// SIMATIC STEP 7 (V5.x) project Q6
// CPU: CPU 313C
// station: Hardware
// station: SIMATIC 300(1)
// station: P_ADR_BUS
// program: S7 Program(1)

SYMBOL_TABLE
"Counter"	C 0	COUNTER
"SCALE"	FC 105	FC 105	// Scaling Values
"UNSCALE"	FC 106	FC 106	// Unscaling Values
"Start"	I 0.0	BOOL
"Stop"	I 0.1	BOOL
"Input Thermocouple"	ID 20	REAL
"Bipolar scale/unscale"	M 0.0	BOOL
"Reserve Motor mem"	M 0.1	BOOL
"MD20"	MD 20	REAL
"Temp INPUT"	MD 30	REAL
"Round Temp INPUT"	MD 50	DINT
"Counter num"	MW 3	INT
"Error Unscale"	MW 10	WORD
"Error Scale"	MW 11	WORD
"Memory OUTPUT"	MW 40	INT
"Buffer"	MW 45	INT
"Out Unscale/IN Scale"	MW 100	INT
"Motor 1"	Q 0.0	BOOL
"Reserve Motor"	Q 0.1	BOOL
"QW100"	QW 100	INT
"Timer"	T 0	TIMER
END_SYMBOL_TABLE

// FC 105: know-how protected block, not included

// FC 106: know-how protected block, not included

ORGANIZATION_BLOCK OB 1
TITLE = "Main Program Sweep (Cycle)"
VERSION : 0.1
VAR_TEMP
  OB1_EV_CLASS : BYTE ;	//Bits 0-3 = 1 (Coming event), Bits 4-7 = 1 (Event class 1)
  OB1_SCAN_1 : BYTE ;	//1 (Cold restart scan 1 of OB 1), 3 (Scan 2-n of OB 1)
  OB1_PRIORITY : BYTE ;	//Priority of OB Execution
  OB1_OB_NUMBR : BYTE ;	//1 (Organization block 1, OB1)
  OB1_RESERVED_1 : BYTE ;	//Reserved for system
  OB1_RESERVED_2 : BYTE ;	//Reserved for system
  OB1_PREV_CYCLE : INT ;	//Cycle time of previous OB1 scan (milliseconds)
  OB1_MIN_CYCLE : INT ;	//Minimum cycle time of OB1 (milliseconds)
  OB1_MAX_CYCLE : INT ;	//Maximum cycle time of OB1 (milliseconds)
  OB1_DATE_TIME : DATE_AND_TIME ;	//Date and time OB1 started
END_VAR
BEGIN
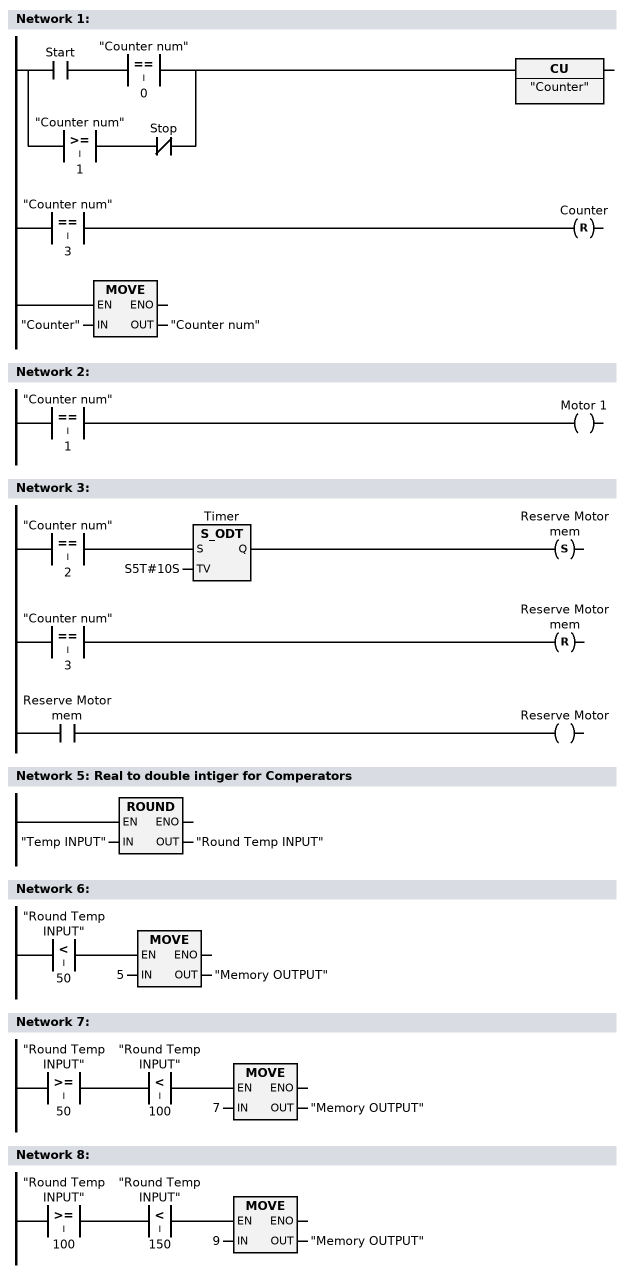
NETWORK
TITLE =
      A(;
      A     "Start";
      A(;
      L     "Counter num";
      L     0;
      ==I;
      );
      O;
      A(;
      L     "Counter num";
      L     1;
      >=I;
      );
      AN    "Stop";
      );
      CU    "Counter";
      BLD   101;
      NOP   0;
      NOP   0;
      A(;
      L     "Counter num";
      L     3;
      ==I;
      );
      R     "Counter";
      L     "Counter";
      T     "Counter num";
      NOP   0;
      NOP   0;
NETWORK
TITLE =
      L     "Counter num";
      L     1;
      ==I;
      =     "Motor 1";
NETWORK
TITLE =
      A(;
      A(;
      L     "Counter num";
      L     2;
      ==I;
      );
      L     S5T#10S;
      SD    "Timer";
      NOP   0;
      NOP   0;
      NOP   0;
      A     "Timer";
      );
      S     "Reserve Motor mem";
      A(;
      L     "Counter num";
      L     3;
      ==I;
      );
      R     "Reserve Motor mem";
      A     "Reserve Motor mem";
      =     "Reserve Motor";
NETWORK
TITLE =
      A     "Bipolar scale/unscale";
      =     L 20.0;
      BLD   103;
      A(;
      A     "Bipolar scale/unscale";
      =     L 20.1;
      BLD   103;
      CALL  "UNSCALE" (
           $1                       := "Input Thermocouple",
           $2                       := L#1101004800,
           $3                       := L#1082130432,
           $4                       := L 20.1,
           $5                       := "Error Unscale",
           $6                       := "Out Unscale/IN Scale");
      A     BR;
      );
      JNB   _001;
      CALL  "SCALE" (
           $1                       := "Out Unscale/IN Scale",
           $2                       := L#1148846080,
           $3                       := L#-1027080192,
           $4                       := L 20.0,
           $5                       := "Error Scale",
           $6                       := "Temp INPUT");
_001: NOP   0;
NETWORK
TITLE = Real to double intiger for Comperators
      L     "Temp INPUT";
      RND;
      T     "Round Temp INPUT";
      NOP   0;
NETWORK
TITLE =
      A(;
      L     "Round Temp INPUT";
      L     50;
      <I;
      );
      JNB   _002;
      L     5;
      T     "Memory OUTPUT";
_002: NOP   0;
NETWORK
TITLE =
      A(;
      L     "Round Temp INPUT";
      L     50;
      >=I;
      );
      A(;
      L     "Round Temp INPUT";
      L     100;
      <I;
      );
      JNB   _003;
      L     7;
      T     "Memory OUTPUT";
_003: NOP   0;
NETWORK
TITLE =
      A(;
      L     "Round Temp INPUT";
      L     100;
      >=I;
      );
      A(;
      L     "Round Temp INPUT";
      L     150;
      <I;
      );
      JNB   _004;
      L     9;
      T     "Memory OUTPUT";
_004: NOP   0;
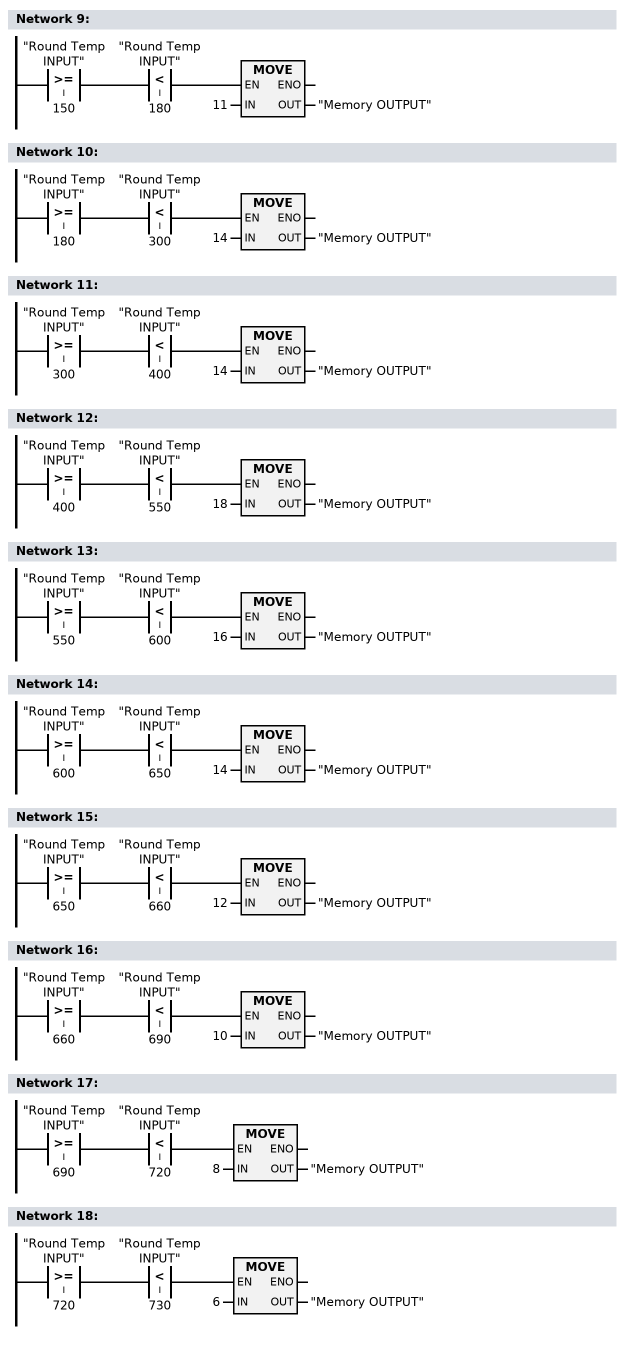
NETWORK
TITLE =
      A(;
      L     "Round Temp INPUT";
      L     150;
      >=I;
      );
      A(;
      L     "Round Temp INPUT";
      L     180;
      <I;
      );
      JNB   _005;
      L     11;
      T     "Memory OUTPUT";
_005: NOP   0;
NETWORK
TITLE =
      A(;
      L     "Round Temp INPUT";
      L     180;
      >=I;
      );
      A(;
      L     "Round Temp INPUT";
      L     300;
      <I;
      );
      JNB   _006;
      L     14;
      T     "Memory OUTPUT";
_006: NOP   0;
NETWORK
TITLE =
      A(;
      L     "Round Temp INPUT";
      L     300;
      >=I;
      );
      A(;
      L     "Round Temp INPUT";
      L     400;
      <I;
      );
      JNB   _007;
      L     14;
      T     "Memory OUTPUT";
_007: NOP   0;
NETWORK
TITLE =
      A(;
      L     "Round Temp INPUT";
      L     400;
      >=I;
      );
      A(;
      L     "Round Temp INPUT";
      L     550;
      <I;
      );
      JNB   _008;
      L     18;
      T     "Memory OUTPUT";
_008: NOP   0;
NETWORK
TITLE =
      A(;
      L     "Round Temp INPUT";
      L     550;
      >=I;
      );
      A(;
      L     "Round Temp INPUT";
      L     600;
      <I;
      );
      JNB   _009;
      L     16;
      T     "Memory OUTPUT";
_009: NOP   0;
NETWORK
TITLE =
      A(;
      L     "Round Temp INPUT";
      L     600;
      >=I;
      );
      A(;
      L     "Round Temp INPUT";
      L     650;
      <I;
      );
      JNB   _00a;
      L     14;
      T     "Memory OUTPUT";
_00a: NOP   0;
NETWORK
TITLE =
      A(;
      L     "Round Temp INPUT";
      L     650;
      >=I;
      );
      A(;
      L     "Round Temp INPUT";
      L     660;
      <I;
      );
      JNB   _00b;
      L     12;
      T     "Memory OUTPUT";
_00b: NOP   0;
NETWORK
TITLE =
      A(;
      L     "Round Temp INPUT";
      L     660;
      >=I;
      );
      A(;
      L     "Round Temp INPUT";
      L     690;
      <I;
      );
      JNB   _00c;
      L     10;
      T     "Memory OUTPUT";
_00c: NOP   0;
NETWORK
TITLE =
      A(;
      L     "Round Temp INPUT";
      L     690;
      >=I;
      );
      A(;
      L     "Round Temp INPUT";
      L     720;
      <I;
      );
      JNB   _00d;
      L     8;
      T     "Memory OUTPUT";
_00d: NOP   0;
NETWORK
TITLE =
      A(;
      L     "Round Temp INPUT";
      L     720;
      >=I;
      );
      A(;
      L     "Round Temp INPUT";
      L     730;
      <I;
      );
      JNB   _00e;
      L     6;
      T     "Memory OUTPUT";
_00e: NOP   0;
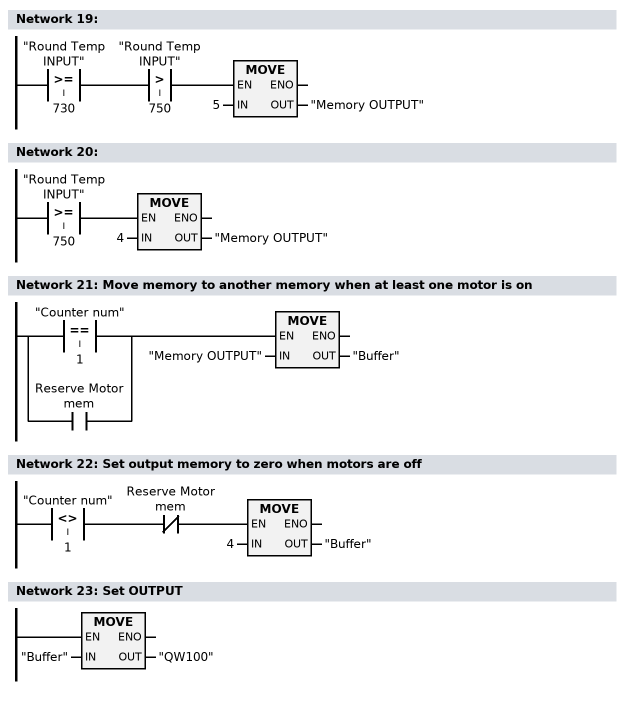
NETWORK
TITLE =
      A(;
      L     "Round Temp INPUT";
      L     730;
      >=I;
      );
      A(;
      L     "Round Temp INPUT";
      L     750;
      >I;
      );
      JNB   _00f;
      L     5;
      T     "Memory OUTPUT";
_00f: NOP   0;
NETWORK
TITLE =
      A(;
      L     "Round Temp INPUT";
      L     750;
      >=I;
      );
      JNB   _010;
      L     4;
      T     "Memory OUTPUT";
_010: NOP   0;
NETWORK
TITLE = Move memory to another memory when at least one motor is on
      A(;
      O(;
      L     "Counter num";
      L     1;
      ==I;
      );
      O     "Reserve Motor mem";
      );
      JNB   _011;
      L     "Memory OUTPUT";
      T     "Buffer";
_011: NOP   0;
NETWORK
TITLE = Set output memory to zero when motors are off
      A(;
      L     "Counter num";
      L     1;
      <>I;
      );
      AN    "Reserve Motor mem";
      JNB   _012;
      L     4;
      T     "Buffer";
_012: NOP   0;
NETWORK
TITLE = Set OUTPUT
      L     "Buffer";
      T     "QW100";
      NOP   0;
END_ORGANIZATION_BLOCK
